# B&R Automation Studio project RTFProj (part 3)

#### Types.typ - Exported data types
```iecst
TYPE
	enum_opticalSensorInternal :
		(
		OS_INITIALIZATION := 0,
		OS_ENABLED := 1,
		OS_CALCULATION := 2,
		OS_ERROR := 3
		);
	struct_opticalSensorInternal : 	STRUCT
		index : ARRAY[0..1]OF USINT;
		auxiliary_pos : ARRAY[0..3]OF REAL;
		state : enum_opticalSensorInternal;
	END_STRUCT;
END_TYPE
```

#### ro_sensors.fun - Exported functions and function blocks
```iecst
FUNCTION err_modDetect : BOOL
	VAR_INPUT
		detect_err : ARRAY[0..3] OF BOOL;
		modul_ok : ARRAY[0..3] OF BOOL;
	END_VAR
	VAR
		i2 : USINT;
		i1 : USINT;
	END_VAR
END_FUNCTION

FUNCTION_BLOCK FB_DetectionPosition
	VAR_INPUT
		Enable : BOOL;
		Distance_Error : ARRAY[0..3] OF BOOL;
		Positions_FromTheSensors : ARRAY[0..3] OF REAL;
		Detection_Error : ARRAY[0..3] OF BOOL;
	END_VAR
	VAR_OUTPUT
		Actual_Positions : ARRAY[0..3] OF REAL;
		ModulOk : ARRAY[0..3] OF BOOL;
		Error : BOOL;
	END_VAR
	VAR
		Internal : struct_opticalSensorInternal;
	END_VAR
END_FUNCTION_BLOCK
```

#### FB_DetectionPosition.st
```iecst
FUNCTION_BLOCK FB_DetectionPosition

    IF Enable <> TRUE THEN
        // reset output variables
        Internal.index[0] := 0;
        Internal.index[1] := 0;

        Actual_Positions[0] := 0;
        Actual_Positions[1] := 0;
        Actual_Positions[2] := 0;
        Actual_Positions[3] := 0;

        ModulOk[0] := FALSE;
        ModulOk[1] := FALSE;
        ModulOk[2] := FALSE;
        ModulOk[3] := FALSE;

        Error := FALSE;

        // go to initialization state
        Internal.state := OS_INITIALIZATION;
    END_IF

    CASE Internal.state OF
        OS_INITIALIZATION:
            // INITIALIZATION STATE
            IF Enable = TRUE THEN
                Internal.state := OS_ENABLED;
            ELSE
                Internal.state := OS_INITIALIZATION;
            END_IF

        OS_ENABLED:
            // ENABLED STATE
            Error := err_modDetect(Detection_Error,ModulOk);

            IF Error = TRUE THEN
                Internal.state := OS_ERROR;
            ELSE
                Internal.state := OS_CALCULATION;
            END_IF

        OS_CALCULATION:
            // CALCULATION STATE
            FOR Internal.index[0] := 0 TO 3 DO
                IF Distance_Error[Internal.index[0]] = FALSE AND Internal.auxiliary_pos[Internal.index[0]] <> -9999 THEN
                    Internal.auxiliary_pos[Internal.index[0]] := 0;
                    Actual_Positions[Internal.index[0]]       := Positions_FromTheSensors[Internal.index[0]];
                ELSIF Distance_Error[Internal.index[0]] = TRUE AND Internal.auxiliary_pos[Internal.index[0]] <> -9999 THEN
                    Internal.auxiliary_pos[Internal.index[0]] := 0;
                    Actual_Positions[Internal.index[0]]       := -1000;
                ELSE
                    Actual_Positions[Internal.index[0]]       := Internal.auxiliary_pos[Internal.index[0]];
                    Internal.auxiliary_pos[Internal.index[0]] := 0;
                END_IF

            END_FOR

            Error := err_modDetect(Detection_Error,ModulOk);

            IF Error = TRUE THEN
                Internal.state := OS_ERROR;
            ELSE
                Internal.state := OS_CALCULATION;
            END_IF
        OS_ERROR:
            // ERROR STATE
            Error := err_modDetect(Detection_Error,ModulOk);

            IF Error = TRUE THEN
                FOR Internal.index[1] := 0 TO 3 DO
                    IF ModulOk[Internal.index[1]] = FALSE THEN
                        Internal.auxiliary_pos[Internal.index[1]] := -9999;
                    ELSE
                        Internal.auxiliary_pos[Internal.index[1]] := 0;
                    END_IF
                END_FOR

                Internal.state := OS_CALCULATION;
            ELSE
                Internal.state := OS_CALCULATION;
            END_IF
    END_CASE

END_FUNCTION_BLOCK

FUNCTION err_modDetect

    FOR i1 := 0 TO 3 DO
        IF detect_err[i1] = FALSE THEN
            modul_ok[i1] := TRUE;
        ELSE
            modul_ok[i1] := FALSE;
        END_IF
    END_FOR

    FOR i2 := 0 TO 3 DO
        IF modul_ok[i2] = FALSE THEN
            err_modDetect := TRUE;
            RETURN;
        ELSE
            err_modDetect := FALSE;
        END_IF
    END_FOR

END_FUNCTION
```

### Library Logical/Libraries/Camera (ANSIC)

#### Types.typ - Exported data types
```iecst
TYPE
	MainSwitch_enum :
		(
		DISABLED := 0,
		ENABLED := 1,
		RUN := 2,
		ERROR := 255
		);
	FTPSwitch_enum :
		(
		DEVLINK := 1,
		FILECOPY := 2,
		DEVUNLINK := 3
		);
	ControlSwitch_enum :
		(
		WAIT_CMD := 0,
		TRIGGER_RDY := 1,
		TRIGGER := 2,
		ACQ := 3,
		INSP := 4
		);
	InSight_type : 	STRUCT
		ModuleOk : BOOL;
		Control_I2000_S01 : UDINT; (*Camera control including trigger*)
		Status_I2001_S01 : UDINT;
		InspectionResults_I2011_S01 : UDINT; (*X Axis*)
		InspectionResults_I2011_S02 : UDINT; (*Y Axis*)
		InspectionResults_I2011_S03 : UDINT; (*Succes*)
		InspectionResults_I2011_S04 : UDINT; (*Fail*)
		UserData_I2021_S01 : UDINT; (*Change zone*)
	END_STRUCT;
	Internal_type : 	STRUCT
		NaN : REAL;
		CameraControl : CameraControl_type;
		MainSwitch : MainSwitch_enum;
		FTP : FTP_type;
		SuccesCount : UDINT;
		FailCount : UDINT;
		disableBit : USINT;
		Search_tmp : BOOL;
		Zone : Zone_enum;
		ChangeZone : ChangeZone_enum;
		oldState : ChangeZone_enum;
	END_STRUCT;
	Zone_enum :
		(
		ZONE1 := 0,
		ZONE2 := 1,
		ZONE3 := 2,
		ZONE4 := 3,
		ZONE5 := 4,
		ZONE6 := 5,
		ZONE7 := 6,
		ZONE8 := 7,
		WHOLE := 500
		);
	ChangeZone_enum :
		(
		CHANGE := 2,
		ONE_ZONE := 1,
		WHOLE_ZONE := 0
		);
	Results_type : 	STRUCT
		AxisX : REAL;
		AxisY : REAL;
		ActTime : RTCtime_typ;
		AxisXOld : REAL;
		AxisYOld : REAL;
		TimeDiff_ms : REAL;
		ActTimeOld : RTCtime_typ;
		NewVal : BOOL;
	END_STRUCT;
	CameraControl_type : 	STRUCT
		ControlSwitch : ControlSwitch_enum;
	END_STRUCT;
	MappView_type : 	STRUCT
		ZoneString : STRING[80];
		PicEnable : BOOL;
		Y : ARRAY[0..1000]OF INT;
		X : ARRAY[0..1000]OF INT := [11(5),0,996(0)];
		LoadImage : BOOL;
	END_STRUCT;
	FTP_type : 	STRUCT
		FileCopy_0 : FileCopy;
		DevLink_0 : DevLink;
		DevUnlink_0 : DevUnlink;
		Status : USINT;
		FTPSwitch : FTPSwitch_enum;
		pParam : STRING[200];
		handle : UDINT;
		pDevice : STRING[20];
		pDest : STRING[80];
		pSrc : STRING[80];
		pDestDev : STRING[20];
	END_STRUCT;
END_TYPE
```

#### Constants.var - Exported constants
```iecst
VAR CONSTANT
	ERR_OK : UINT := 0;
	FB_DISABLED : UINT := 65534; (*Function block is disabled*)
	ERR_CAM_NOTFOUND : UINT := 65533; (*Camera not found*)
	ERR_FTP_NOTREADY : UINT := 62687; (*FTP not ready*)
END_VAR
```

#### Camera.fun - Exported functions and function blocks
```iecst
FUNCTION_BLOCK FBCamera
	VAR_INPUT
		Enable : BOOL;
		InSight : InSight_type;
		ErrorReset : BOOL;
		Search : BOOL;
	END_VAR
	VAR_OUTPUT
		Active : BOOL;
		Error : BOOL;
		Status : UINT;
		isCameraReady : BOOL;
		isSearching : BOOL;
		isBallFound : BOOL;
		Results : Results_type;
	END_VAR
	VAR
		Internal : Internal_type;
	END_VAR
END_FUNCTION_BLOCK
```

#### Camera.c
```c
#include <bur/plctypes.h>
#include <math.h>

#ifdef _DEFAULT_INCLUDES
#include <AsDefault.h>
#endif

#define NaN sqrt(-1)
#define CAM_OFFLINE_MASK 128												//1000 0000b
#define CAM_ONLINE_MASK 0xFFFFFF7F

#define CAM_USER_DATA 0x10004												//Mask for user data ack
#define CAM_FIND_WHOLE_ZONE 0xFFFFFFFF										//Mask for finding at whole playground

#define MAX_DIFF_PER 0.15													//Max diffrence between old and actual value in %

#define ABS_F(X) ((X) < (0) ? -(X) : (X)) 									//ABS funkcion
							//		  |							9800
#define X1_REF_PLGND 800.0	//(UNITS) |				   3800 6800  | 11300
#define X2_REF_PLGND 11300.0//(UNITS) |				 _____|___|___|_|_
#define X1_REF_CAM 1215.0	//(PIXELS)|				| | | O O O O | | |		SCHEME OF X AXIS
#define X2_REF_CAM 82.0		//(PIXELS)|				| | O | O O | O | |		AND PLAYGROUND WITH
 							//		  |		    	| O | O O O O | O |		DISTANCE OF PLAYERS
#define Y1_REF_PLGND 820.0	//(UNITS) |	 	  		| | O | O O | O | |		IN UNITS
#define Y2_REF_PLGND -950.0 //(UNITS) |				|_|_|_O_O_O_O_|_|_|		(10 UNITS = 1 MM)
#define Y1_REF_CAM 414.0	//(PIXELS)| 		      | |   |   |
#define Y2_REF_CAM 604.0	//(PIXELS)|			 	800 | 5300 8300
							//		  |		    	   2300

#define X_LIN_EQ_K ((X1_REF_PLGND-X2_REF_PLGND)/(X1_REF_CAM-X2_REF_CAM)) 		//Define K-parameter of line equaton for X axis
#define X_LIN_EQ_Q (X1_REF_PLGND-(X1_REF_CAM*X_LIN_EQ_K))				 		//Define Q-parameter of line equaion for X axis

#define Y_LIN_EQ_K ((Y1_REF_PLGND-Y2_REF_PLGND)/(Y1_REF_CAM-Y2_REF_CAM))		//Define K-parameter of line equaton for Y axis
#define Y_LIN_EQ_Q (Y1_REF_PLGND-(Y1_REF_CAM*Y_LIN_EQ_K))						//Define Q-parameter of line equaton for Y axis

#define X_MAX_DIFF ABS_F((X_LIN_EQ_K+X_LIN_EQ_Q)-((2*X_LIN_EQ_K)+X_LIN_EQ_Q))	//Line equation for X axis
#define Y_MAX_DIFF ABS_F((Y_LIN_EQ_K+Y_LIN_EQ_Q)-((2*Y_LIN_EQ_K)+Y_LIN_EQ_Q))	//Line equation for Y axis

void setError(struct FBCamera *inst,unsigned int status);
void initFB(struct FBCamera *inst);
void resetFB(struct FBCamera *inst);
void getRealAxes(struct FBCamera *inst);
void cleanFB(struct FBCamera *inst);
REAL RctToReal_ms (struct RTCtime_typ RTCtime);

void FBCamera(struct FBCamera *inst)
{
	if ((!inst->Enable) && (!inst->Internal.disableBit))
		cleanFB(inst);

	switch (inst->Internal.MainSwitch){										//Main switch, DISABLED FB, INITialising FB, ENABLED FB and ERROR case
		/******************************************************************/
		/*							FB is DISABLED					 	  */
		/******************************************************************/

		case DISABLED:														//FB is disabled
			if (inst->Internal.disableBit){
				cleanFB(inst);
				inst->Internal.disableBit = 1;
			}
			if (inst->Enable){												//Wait for Enable = TRUE, else do nothing
				inst->Internal.MainSwitch = ENABLED;						//Go to ENABLED case
				inst->Internal.disableBit = 0;
			}
			else
				inst->Status = ERR_FUB_ENABLE_FALSE;						//Status 65534, FB is called but not enabled
			break;

		/******************************************************************/
		/*				FB is ENABLED but Camera is not ready		 	  */
		/******************************************************************/

		case ENABLED:														//FB is enabled and working
			inst->Status = ERR_OK;											//No error in enable case
			inst->Active = 1;												//variable indicating active FB
			if (!inst->InSight.ModuleOk){									//InSight Camera is not connected properly
				inst->isCameraReady = 0;									//Bit for user that Camera is not working
				if (inst->Search)											//If user allow searching for ball, change case to ERROR because you cannot find while there is no camera
					setError(inst,ERR_CAM_NOTFOUND);						//Error, Status 65533 - camera not found
			}
			else {
				inst->isCameraReady = 1;									//Bit for user that Camera is working
				inst->Internal.MainSwitch = RUN;							//Change state to RUN
			}
			break;

		/******************************************************************/
		/*						FB and Camera are ready				 	  */
		/******************************************************************/
		case RUN:															//FB is enabled and camera communicating
			if (!(inst->InSight.ModuleOk))									//if camera is disconnected change state to ENABLE where waiting for connect
				inst->Internal.MainSwitch = ENABLED;
			if (inst->Search){
				inst->isSearching = 1;
				inst->InSight.Control_I2000_S01 &= CAM_ONLINE_MASK;			//Disable control bit for cammera offline mode
				switch (inst->Internal.ChangeZone){
					case CHANGE:
						if ((inst->InSight.Control_I2000_S01 & CAM_USER_DATA) == CAM_USER_DATA){
							if ((inst->InSight.Status_I2001_S01 & 0x10000) == 0x10000) {
								if (inst->Internal.oldState == ONE_ZONE)
									inst->Internal.ChangeZone = WHOLE_ZONE;
								else
									inst->Internal.ChangeZone = ONE_ZONE;
								inst->InSight.Control_I2000_S01 &= 0xFFFEFFFB;
							}
						}
						else inst->Internal.ChangeZone = WHOLE_ZONE;
						break;

					case ONE_ZONE:
						getRealAxes(inst);
						inst->Internal.oldState = ONE_ZONE;
						if (((isnan(inst->Results.AxisX)) || isnan(inst->Results.AxisY)) && (inst->Results.NewVal)){
							inst->Internal.ChangeZone = CHANGE;
							inst->InSight.Control_I2000_S01 |= CAM_USER_DATA;
							inst->InSight.UserData_I2021_S01 = 65535;
						}
						switch (inst->Internal.Zone){
							case ZONE1:
								strcpy(inst->MappView.ZoneString,"Zone 1");
								break;

							case ZONE2:
								strcpy(inst->MappView.ZoneString,"Zone 2");
								break;

							case ZONE3:
								strcpy(inst->MappView.ZoneString,"Zone 3");
								break;

							case ZONE4:
								strcpy(inst->MappView.ZoneString,"Zone 4");
								break;

							case ZONE5:
								strcpy(inst->MappView.ZoneString,"Zone 5");
								break;

							case ZONE6:
								strcpy(inst->MappView.ZoneString,"Zone 6");
								break;

							case ZONE7:
								strcpy(inst->MappView.ZoneString,"Zone 7");
								break;

							case WHOLE:

								break;
						}
						break;

					case WHOLE_ZONE:
						getRealAxes(inst);
						inst->Internal.Zone = WHOLE;
						inst->Internal.oldState = WHOLE_ZONE;
						strcpy(inst->MappView.ZoneString,"Whole");
						if(inst->isBallFound){
							inst->Internal.ChangeZone = CHANGE;
							inst->InSight.Control_I2000_S01 |= CAM_USER_DATA;
							if (inst->Results.AxisX > 10300){
								inst->InSight.UserData_I2021_S01 = 1;
								inst->Internal.Zone = ZONE1;}
							else if (inst->Results.AxisX > 9050){
								inst->InSight.UserData_I2021_S01 = 2;
								inst->Internal.Zone = ZONE2;}
							else if (inst->Results.AxisX > 7350){
								inst->InSight.UserData_I2021_S01 = 4;
								inst->Internal.Zone = ZONE3;}
							else if (inst->Results.AxisX > 6250){
								inst->InSight.UserData_I2021_S01 = 8;
								inst->Internal.Zone = ZONE4;}
							else if (inst->Results.AxisX > 4400){
								inst->InSight.UserData_I2021_S01 = 16;
								inst->Internal.Zone = ZONE5;}
							else if (inst->Results.AxisX > 2460){
								inst->InSight.UserData_I2021_S01 = 32;
								inst->Internal.Zone = ZONE6;}
							else if (inst->Results.AxisX > 0){
								inst->InSight.UserData_I2021_S01 = 64;
								inst->Internal.Zone = ZONE7;}
							else{
								inst->Internal.ChangeZone = WHOLE_ZONE;
								inst->InSight.Control_I2000_S01 &= 0xFFFEFFFB;
								inst->InSight.UserData_I2021_S01 = 0xFFFF;
							}
						}
						break;

				}
			}
			else{
				inst->InSight.Control_I2000_S01 |= CAM_OFFLINE_MASK;
				inst->isSearching = 0;
			}
			break;

		case ERROR:															//error case, to change state is needed error Reset variable or disable FB
			inst->Error = 1;												//Change Error variable
			inst->Internal.CameraControl.ControlSwitch = WAIT_CMD;			//Reset camera trigger state
			inst->isSearching = 0;											//FB cannot searching in error case
			if (inst->ErrorReset){											//waiting on ErrorReset
				inst->Error = 0;
				inst->Status = ERR_OK;
				resetFB(inst);
				inst->Internal.MainSwitch = ENABLED;						//change state
			}
			break;
	}

	if (inst->ErrorReset)
		resetFB(inst);

	if (inst->Error == 1)
		inst->Internal.MainSwitch = ERROR;

}

void initFB(struct FBCamera *inst)
{
	inst->Active = 0;
	inst->Error = 0;
	inst->ErrorReset = 0;
	inst->isCameraReady = 0;
	inst->isBallFound = 0;
	inst->isSearching = 0;
	inst->Search = 0;
	inst->Status = ERR_OK;
	inst->Internal.CameraControl.ControlSwitch = WAIT_CMD;
	inst->Internal.MainSwitch = DISABLED;
	inst->Internal.Search_tmp = 0;
	inst->Internal.disableBit = 1;
	inst->InSight.Control_I2000_S01 |= CAM_OFFLINE_MASK;
	memset(&inst->Results.ActTime,0,sizeof(inst->Results.ActTime));
	inst->Results.AxisXOld = NaN;
	inst->Results.AxisYOld = NaN;
	inst->InSight.Control_I2000_S01 |= CAM_USER_DATA;
	inst->InSight.UserData_I2021_S01 = 65535;
	inst->Internal.ChangeZone = CHANGE;
}

void resetFB(struct FBCamera *inst)
{
	inst->ErrorReset = 0;							//Reset error reset
	inst->Error = 0;								//Reset Error
	inst->Status = ERR_OK;
}

void cleanFB(struct FBCamera *inst)
{
	initFB(inst);
	resetFB(inst);
}

void setError(struct FBCamera *inst,unsigned int status) {
	inst->Error = 1;
	inst->Status = status;
}

void getRealAxes(struct FBCamera *inst)
{
	if (inst->Internal.SuccesCount != inst->InSight.InspectionResults_I2011_S03){
		inst->Results.NewVal = 1;
		REAL AxisXnew = ((inst->InSight.InspectionResults_I2011_S01*X_LIN_EQ_K)+X_LIN_EQ_Q);
		REAL AxisYnew = ((inst->InSight.InspectionResults_I2011_S02*Y_LIN_EQ_K)+Y_LIN_EQ_Q);

		if (((AxisXnew >= 0) && (AxisXnew < 12100)) && ((AxisYnew < 3515) && (AxisYnew > -3515))){

			if (isnan(inst->Results.AxisX) || isnan(inst->Results.AxisY)){
				inst->Results.AxisX = AxisXnew;
				inst->Results.AxisY = AxisYnew;
			}
			else if(((ABS_F(AxisXnew - (inst->Results.AxisX))) < (X_MAX_DIFF * 2)) && (((ABS_F(AxisYnew - (inst->Results.AxisY))) < (Y_MAX_DIFF * 2)))) {
				inst->Results.AxisXOld = inst->Results.AxisX = ((AxisXnew + inst->Results.AxisX)/2);
				inst->Results.AxisYOld = inst->Results.AxisY = ((AxisYnew + inst->Results.AxisY)/2);
			}
			else{
				inst->Results.AxisXOld = inst->Results.AxisX;
				inst->Results.AxisYOld = inst->Results.AxisY;
				inst->Results.AxisX = AxisXnew;
				inst->Results.AxisY = AxisYnew;
			}
			memcpy((UDINT)&inst->Results.ActTimeOld,(UDINT)&inst->Results.ActTime,sizeof(inst->Results.ActTime));
			RTC_gettime(&inst->Results.ActTime);
			inst->Results.TimeDiff_ms = ((RctToReal_ms(inst->Results.ActTime)) - (RctToReal_ms(inst->Results.ActTimeOld)));
			inst->isBallFound = 1;
			inst->Status = ERR_OK;
			inst->Internal.SuccesCount = inst->InSight.InspectionResults_I2011_S03;
		}
		else{
			inst->Status = ERR_BALL_OUTRANGE;
			inst->isBallFound = 0;
		}
	}
	else if (inst->Internal.FailCount != inst->InSight.InspectionResults_I2011_S04){
		inst->Results.NewVal = 1;
		if (!isnan(inst->Results.AxisX) || !isnan(inst->Results.AxisY)){
			inst->Results.AxisXOld = inst->Results.AxisX;
			inst->Results.AxisYOld = inst->Results.AxisY;
		}
		inst->Results.AxisX = inst->Results.AxisY = NaN;
		inst->Internal.FailCount = inst->InSight.InspectionResults_I2011_S04;
		inst->isBallFound = 0;
		memcpy((UDINT)&inst->Results.ActTimeOld,(UDINT)&inst->Results.ActTime,sizeof(inst->Results.ActTime));
		RTC_gettime(&inst->Results.ActTime);
		inst->Results.TimeDiff_ms = ((RctToReal_ms(inst->Results.ActTime)) - (RctToReal_ms(inst->Results.ActTimeOld)));
	}
	else{
		inst->isBallFound = 0;
		inst->Results.NewVal = 1;
	}
}

REAL RctToReal_ms (struct RTCtime_typ RTCtime){
	return(((REAL)RTCtime.hour*3600000)+((REAL)RTCtime.minute*60000)+((REAL)RTCtime.second*1000)+((REAL)RTCtime.millisec)+((REAL)RTCtime.microsec/1000));
}
```

### Library Logical/Libraries/Bar_Light (ANSIC)

#### Bar_light.c
```c
#include <bur/plctypes.h>
#include <MTBasics.h>
#include <brsystem.h>
#include <math.h>

#ifdef _DEFAULT_INCLUDES
#include <AsDefault.h>
#endif

void resetFB(struct Light *inst);												//Reset basic variables
void PWMControl(struct Light *inst);											//Controls Light in PWM Mode
void BlinkControl(struct Light *inst);											//Allows Blinking of Light

void Light(struct Light *inst)
{
	if ((!inst->Enable) && (inst->internal.MainControlBarLight != INIT_BARLIGHT))//If FB not allowed and switch is not in init state
		inst->internal.MainControlBarLight = DISABLED_BARLIGHT;					//Change state to DISABLED

	switch (inst->internal.MainControlBarLight)									//Main switch controls whole FB
	{
		case INIT_BARLIGHT:														//Check parameter for PWM
			inst->internal.TaskClass.RTInfo_0.enable = 1;
			RTInfo(&inst->internal.TaskClass.RTInfo_0);
			if (!(inst->internal.TaskClass.RTInfo_0.status) && (inst->internal.TaskClass.RTInfo_0.cycle_time > 0))
			{
				if (inst->internal.TaskClass.RTInfo_0.cycle_time <= 1000)
				{
					inst->isPWMEnabled = inst->internal.PWM.PWMEnabled = 1;
					inst->isPWMEnabled = inst->internal.PWM.PWM.Enable = 1;
					inst->internal.PWM.PWM.MinPulseWidth = 0.001;
					inst->internal.PWM.PWM.Period = 0.01;
					inst->internal.PWM.PWM.Mode = mtBASICS_PULSE_BEGINNING;
				}
				else
					inst->isPWMEnabled = inst->internal.PWM.PWMEnabled = 0;

				inst->internal.PWM.PWM.DutyCycle = 100;
				inst->internal.TaskClass.RTInfo_0.enable = 0;
				inst->internal.TaskClass.CyclicTime = ((inst->internal.TaskClass.RTInfo_0.cycle_time)/1000);
				inst->internal.MainControlBarLight = DISABLED_BARLIGHT;
			}
			break;

		case DISABLED_BARLIGHT:
			if (inst->Enable)
			{
				if (inst->DO9322.ModuleOK)
				{
					inst->internal.MainControlBarLight = ENABLED_BARLIGHT;
					resetFB(inst);
				}
				else
				{
					inst->Status = DO9322_NOT_CONNECTED;
					inst->internal.MainControlBarLight = ERROR_BARLIGHT;
				}
			}
			break;

		case ENABLED_BARLIGHT:
			inst->Active = 1;
			if (inst->PowerOn)
			{
				if (inst->Blinking.StartBlinking)
				{
					BlinkControl(inst);
				}
				else if (inst->internal.PWM.PWMEnabled)
				{
					PWMControl(inst);
				}
				else inst->DO9322.DigitalOutput = 1;
			}
			else inst->DO9322.DigitalOutput = 0;
			break;

		case ERROR_BARLIGHT:
			inst->Error = 1;
			break;
	}
}

void resetFB(struct Light *inst)
{
	inst->Active = 0;
	inst->Blinking.StartBlinking = 0;
	inst->DO9322.DigitalOutput = 0;
	inst->DutyCycle = 100;
	inst->Error = 0;
	inst->PowerOn = 0;
	inst->isPowerOn = 0;
	inst->Status = ERR_OK;
}

void PWMControl(struct Light *inst)
{
	inst->internal.PWM.PWM.DutyCycle = inst->DutyCycle;
	MTBasicsPWM(&inst->internal.PWM.PWM);
	inst->DO9322.DigitalOutput = inst->internal.PWM.PWM.Out;
}

void BlinkControl(struct Light *inst)
{
	inst->internal.BlinkingCounter += 1;
	if ((inst->internal.BlinkingCounter*inst->internal.TaskClass.CyclicTime) < inst->Blinking.BlinkingTime_ms)
	{
		if ((inst->internal.BlinkCounter*inst->internal.TaskClass.CyclicTime) >= inst->Blinking.BlinkPeriod_ms)
		{
			inst->DO9322.DigitalOutput = !inst->DO9322.DigitalOutput;
			inst->internal.BlinkCounter = 0;
		}
		else
		{
			inst->internal.BlinkCounter += 1;
		}
	}
	else
	{
		inst->internal.BlinkingCounter = 0;
		inst->internal.BlinkCounter = 0;
		inst->DO9322.DigitalOutput = 0;
		inst->Blinking.StartBlinking = 0;
	}
}
```

### Library Logical/Libraries/LB_Camera/Camera (ANSIC)

#### Camera.c
```c
#include <bur/plctypes.h>
#include <math.h>

#ifdef _DEFAULT_INCLUDES
#include <AsDefault.h>
#endif

#define NaN sqrt(-1)
#define CAM_OFFLINE_MASK 128												//1000 0000b
#define CAM_ONLINE_MASK 0xFFFFFF7F

#define ABS_F(X) ((X) < (0) ? -(X) : (X)) 									//ABS funkcion
							//		  |							9800
#define X1_REF_PLGND 800.0	//(UNITS) |				   3800 6800  | 11300
#define X2_REF_PLGND 11300.0//(UNITS) |				 _____|___|___|_|_
#define X1_REF_CAM 1215.0	//(PIXELS)|				| | | O O O O | | |		SCHEME OF X AXIS
#define X2_REF_CAM 82.0		//(PIXELS)|				| | O | O O | O | |		AND PLAYGROUND WITH
 							//		  |		    	| O | O O O O | O |		DISTANCE OF PLAYERS
#define Y1_REF_PLGND 820.0	//(UNITS) |	 	  		| | O | O O | O | |		IN UNITS
#define Y2_REF_PLGND -950.0 //(UNITS) |				|_|_|_O_O_O_O_|_|_|		(10 UNITS = 1 MM)
#define Y1_REF_CAM 414.0	//(PIXELS)| 		      | |   |   |
#define Y2_REF_CAM 604.0	//(PIXELS)|			 	800 | 5300 8300
							//		  |		    	   2300

#define X_LIN_EQ_K ((X1_REF_PLGND-X2_REF_PLGND)/(X1_REF_CAM-X2_REF_CAM)) 		//Define K-parameter of line equaton for X axis
#define X_LIN_EQ_Q (X1_REF_PLGND-(X1_REF_CAM*X_LIN_EQ_K))				 		//Define Q-parameter of line equaion for X axis

#define Y_LIN_EQ_K ((Y1_REF_PLGND-Y2_REF_PLGND)/(Y1_REF_CAM-Y2_REF_CAM))		//Define K-parameter of line equaton for Y axis
#define Y_LIN_EQ_Q (Y1_REF_PLGND-(Y1_REF_CAM*Y_LIN_EQ_K))						//Define Q-parameter of line equaton for Y axis

#define X_MAX_DIFF ABS_F((X_LIN_EQ_K+X_LIN_EQ_Q)-((2*X_LIN_EQ_K)+X_LIN_EQ_Q))	//Line equation for X axis
#define Y_MAX_DIFF ABS_F((Y_LIN_EQ_K+Y_LIN_EQ_Q)-((2*Y_LIN_EQ_K)+Y_LIN_EQ_Q))	//Line equation for Y axis

void setError(struct FBCamera *inst,unsigned int status);
void initFB(struct FBCamera *inst);
void resetFB(struct FBCamera *inst);
void getRealAxes(struct FBCamera *inst);
void cleanFB(struct FBCamera *inst);
REAL RctToReal_ms (struct RTCtime_typ RTCtime);

void FBCamera(struct FBCamera *inst)
{
	if ((!inst->Enable) && (!inst->Internal.disableBit))
		cleanFB(inst);

	switch (inst->Internal.MainSwitch){										//Main switch, DISABLED FB, INITialising FB, ENABLED FB and ERROR case
		/******************************************************************/
		/*							FB is DISABLED					 	  */
		/******************************************************************/

		case DISABLED:														//FB is disabled
			if (inst->Internal.disableBit){
				cleanFB(inst);
				inst->Internal.disableBit = 1;
			}
			if (inst->Enable){												//Wait for Enable = TRUE, else do nothing
				inst->Internal.MainSwitch = ENABLED;						//Go to ENABLED case
				inst->Internal.disableBit = 0;
			}
			else
				inst->Status = ERR_FUB_ENABLE_FALSE;						//Status 65534, FB is called but not enabled
			break;

		/******************************************************************/
		/*				FB is ENABLED but Camera is not ready		 	  */
		/******************************************************************/

		case ENABLED:														//FB is enabled and working
			inst->Active = 1;												//variable indicating active FB
			if (!inst->InSight.ModuleOk){									//InSight Camera is not connected properly
				inst->isCameraReady = 0;									//Bit for user that Camera is not working
				if (inst->Search)											//If user allow searching for ball, change case to ERROR because you cannot find while there is no camera
					setError(inst,ERR_CAM_NOTFOUND);						//Error, Status 65533 - camera not found
			}
			else {
				unsigned int status;
				inst->isCameraReady = 1;								//Bit for user that Camera is working
				inst->Internal.MainSwitch = RUN;						//Change state to RUN
				inst->Status = ERR_OK;									//No error in enable case
			}
			break;

		case RUN:															//FB is enabled and camera communicating
			if (!(inst->InSight.ModuleOk))									//if camera is disconnected change state to ENABLE where waiting for connect
				inst->Internal.MainSwitch = ENABLED;
			if (inst->Search){
				inst->InSight.Control_I2000_S01 &= CAM_ONLINE_MASK;			//Disable control bit for cammera offline mode
				inst->isSearching = 1;
				if (inst->InSight.InspectionResults_I2011_S03 != inst->Internal.SuccesCount)
					inst->isBallFound = 1;
				else inst->isBallFound = 0;
				getRealAxes(inst);
			}
			else{
				inst->InSight.Control_I2000_S01 |= CAM_OFFLINE_MASK;
				inst->isSearching = 0;
			}
			break;

		case ERROR:															//error case, to change state is needed error Reset variable or disable FB
			inst->Error = 1;												//Change Error variable
			inst->Internal.CameraControl.ControlSwitch = WAIT_CMD;			//Reset camera trigger state
			inst->isSearching = 0;											//FB cannot searching in error case
			if (inst->ErrorReset){											//waiting on ErrorReset
				inst->Error = 0;
				inst->Status = ERR_OK;
				resetFB(inst);
				inst->Internal.MainSwitch = ENABLED;						//change state
			}
			break;
	}

	if (inst->ErrorReset)
		resetFB(inst);

	if (inst->Error == 1)
		inst->Internal.MainSwitch = ERROR;

}

void initFB(struct FBCamera *inst)
{
	inst->Active = 0;
	inst->Error = 0;
	inst->ErrorReset = 0;
	inst->isCameraReady = 0;
	inst->isBallFound = 0;
	inst->isSearching = 0;
	inst->Search = 0;
	inst->Status = ERR_OK;
	inst->Internal.CameraControl.ControlSwitch = WAIT_CMD;
	inst->Internal.MainSwitch = DISABLED;
	inst->Internal.Search_tmp = 0;
	inst->Internal.disableBit = 1;
	inst->InSight.Control_I2000_S01 |= CAM_OFFLINE_MASK;
	memset(&inst->Results.ActTime,0,sizeof(inst->Results.ActTime));
	inst->Results.AxisXOld = NaN;
	inst->Results.AxisYOld = NaN;
}

void resetFB(struct FBCamera *inst)
{
	inst->ErrorReset = 0;							//Reset error reset
	inst->Error = 0;								//Reset Error
	inst->Status = ERR_OK;
}

void cleanFB(struct FBCamera *inst)
{
	initFB(inst);
	resetFB(inst);
}

void setError(struct FBCamera *inst,unsigned int status) {
	inst->Error = 1;
	inst->Status = status;
}

void getRealAxes(struct FBCamera *inst)
{
	if (inst->Internal.SuccesCount != inst->InSight.InspectionResults_I2011_S03){
		if(((ABS_F(((inst->InSight.InspectionResults_I2011_S01*X_LIN_EQ_K)+X_LIN_EQ_Q)-(inst->Results.AxisX))) < (X_MAX_DIFF + (0.1*X_MAX_DIFF))) &&
		((ABS_F(((inst->InSight.InspectionResults_I2011_S02*Y_LIN_EQ_K)+Y_LIN_EQ_Q)-(inst->Results.AxisY))) < (Y_MAX_DIFF + (0.1*Y_MAX_DIFF)))) {
			inst->Results.AxisX = ((((inst->InSight.InspectionResults_I2011_S01*(X_LIN_EQ_K))+X_LIN_EQ_Q)+inst->Results.AxisX)/2);
			inst->Results.AxisY = ((((inst->InSight.InspectionResults_I2011_S02*(Y_LIN_EQ_K))+Y_LIN_EQ_Q)+inst->Results.AxisY)/2);
			inst->Results.AxisXOld = inst->Results.AxisYOld = NaN;
		}
		else{
			inst->Results.AxisXOld = inst->Results.AxisX;
			inst->Results.AxisYOld = inst->Results.AxisY;
			inst->Results.AxisX = ((inst->InSight.InspectionResults_I2011_S01*(X_LIN_EQ_K))+X_LIN_EQ_Q);
			inst->Results.AxisY = ((inst->InSight.InspectionResults_I2011_S02*(Y_LIN_EQ_K))+Y_LIN_EQ_Q);

		}
		memcpy((UDINT)&inst->Results.ActTimeOld,(UDINT)&inst->Results.ActTime,sizeof(inst->Results.ActTime));
		RTC_gettime(&inst->Results.ActTime);
		inst->Results.TimeDiff_ms = ((RctToReal_ms(inst->Results.ActTime)) - (RctToReal_ms(inst->Results.ActTimeOld)));
		inst->isBallFound = 1;
		inst->Internal.SuccesCount = inst->InSight.InspectionResults_I2011_S03;
	}
	else if ((inst->Internal.FailCount != inst->InSight.InspectionResults_I2011_S04) && ((!isnan(inst->Results.AxisXOld)) && (!isnan(inst->Results.AxisYOld)))){
		inst->Results.AxisX = inst->Results.AxisXOld;
		inst->Results.AxisY = inst->Results.AxisYOld;
		inst->Results.AxisXOld = inst->Results.AxisYOld = NaN;
		inst->Internal.FailCount = inst->InSight.InspectionResults_I2011_S04;
		inst->isBallFound = 0;
	}
}

REAL RctToReal_ms (struct RTCtime_typ RTCtime){
	return(((REAL)RTCtime.hour*3600000)+((REAL)RTCtime.minute*60000)+((REAL)RTCtime.second*1000)+((REAL)RTCtime.millisec)+((REAL)RTCtime.microsec/1000));
}
```

#### Types.typ - Exported data types
```iecst
TYPE
	MainSwitch_enum :
		(
		DISABLED := 0,
		ENABLED := 1,
		RUN := 2,
		ERROR := 255
		);
	FTPSwitch_enum :
		(
		DEVLINK := 1,
		FILECOPY := 2,
		DEVUNLINK := 3
		);
	ControlSwitch_enum :
		(
		WAIT_CMD := 0,
		TRIGGER_RDY := 1,
		TRIGGER := 2,
		ACQ := 3,
		INSP := 4
		);
	InSight_type : 	STRUCT
		ModuleOk : BOOL;
		Control_I2000_S01 : UDINT; (*Camera control including trigger*)
		Status_I2001_S01 : UDINT;
		InspectionResults_I2011_S02 : UDINT;
		InspectionResults_I2011_S01 : UDINT;
	END_STRUCT;
	Internal_type : 	STRUCT
		NaN : REAL;
		CameraControl : CameraControl_type;
		MainSwitch : MainSwitch_enum;
		FTP : FTP_type;
		disableBit : USINT;
		Search_tmp : BOOL;
	END_STRUCT;
	Results_type : 	STRUCT
		AxisX : REAL;
		AxisY : REAL;
		ActTime : RTCtime_typ;
		AxisXOld : REAL;
		AxisYOld : REAL;
		TimeDiff : REAL;
		ActTimeOld : RTCtime_typ;
	END_STRUCT;
	CameraControl_type : 	STRUCT
		ControlSwitch : ControlSwitch_enum;
	END_STRUCT;
	MappView_type : 	STRUCT
		PicEnable : BOOL;
		Y : ARRAY[0..1000]OF INT;
		X : ARRAY[0..1000]OF INT := [11(5),0,996(0)];
		LoadImage : BOOL;
	END_STRUCT;
	FTP_type : 	STRUCT
		FileCopy_0 : FileCopy;
		DevLink_0 : DevLink;
		DevUnlink_0 : DevUnlink;
		Status : USINT;
		FTPSwitch : FTPSwitch_enum;
		pParam : STRING[200];
		handle : UDINT;
		pDevice : STRING[20];
		pDest : STRING[80];
		pSrc : STRING[80];
		pDestDev : STRING[20];
	END_STRUCT;
END_TYPE
```

#### Constants.var - Exported constants
```iecst
VAR CONSTANT
	ERR_OK : UINT := 0;
	FB_DISABLED : UINT := 65534; (*Function block is disabled*)
	ERR_CAM_NOTFOUND : UINT := 65533; (*Camera not found*)
END_VAR
```

### Library Logical/Libraries/LB_Camera/Bar_Light (ANSIC)
Depends on: MTBasics, brsystem

#### Bar_light.c
```c
#include <bur/plctypes.h>
#include <MTBasics.h>
#include <brsystem.h>
#include <math.h>

#ifdef _DEFAULT_INCLUDES
#include <AsDefault.h>
#endif

void resetFB(struct Light *inst);
void PWMControl(struct Light *inst);
void BlinkControl(struct Light *inst);

void Light(struct Light *inst)
{
	if ((!inst->Enable) && (inst->internal.MainControlBarLight != INIT_BARLIGHT))
	{
		inst->internal.MainControlBarLight = DISABLED_BARLIGHT;
	}

	switch (inst->internal.MainControlBarLight)
	{
		case INIT_BARLIGHT:
			inst->internal.TaskClass.RTInfo_0.enable = 1;
			RTInfo(&inst->internal.TaskClass.RTInfo_0);
			if (!(inst->internal.TaskClass.RTInfo_0.status) && (inst->internal.TaskClass.RTInfo_0.cycle_time > 0))
			{
				if (inst->internal.TaskClass.RTInfo_0.cycle_time <= 1000)
				{
					inst->isPWMEnabled = inst->internal.PWM.PWMEnabled = 1;
					inst->internal.PWM.PWM.MinPulseWidth = 0.001;
					inst->internal.PWM.PWM.Period = 0.1;
					inst->internal.PWM.PWM.Mode = mtBASICS_PULSE_BEGINNING;
				}
				else
					inst->isPWMEnabled = inst->internal.PWM.PWMEnabled = 0;

				inst->internal.PWM.PWM.DutyCycle = 100;
				inst->internal.TaskClass.RTInfo_0.enable = 0;
				inst->internal.TaskClass.CyclicTime = ((inst->internal.TaskClass.RTInfo_0.cycle_time)/1000);
				inst->internal.MainControlBarLight = DISABLED_BARLIGHT;
			}
			break;

		case DISABLED_BARLIGHT:
			if (inst->Enable)
			{
				if (inst->DO9322.ModuleOK)
				{
					inst->internal.MainControlBarLight = ENABLED_BARLIGHT;
					resetFB(inst);
				}
				else
				{
					inst->Status = DO9322_NOT_CONNECTED;
					inst->internal.MainControlBarLight = ERROR_BARLIGHT;
				}
			}
			break;

		case ENABLED_BARLIGHT:
			inst->Active = 1;
			if (inst->PowerOn)
			{
				if (inst->Blinking.StartBlinking)
				{
					BlinkControl(inst);
				}
				else if (inst->internal.PWM.PWMEnabled)
				{
					PWMControl(inst);
				}
				else inst->DO9322.DigitalOutput = 1;
			}
			else inst->DO9322.DigitalOutput = 0;
			break;

		case ERROR_BARLIGHT:
			inst->Error = 1;
			break;
	}
}

void resetFB(struct Light *inst)
{
	inst->Active = 0;
	inst->Blinking.StartBlinking = 0;
	inst->DO9322.DigitalOutput = 0;
	inst->DutyCycle = 100;
	inst->Error = 0;
	inst->PowerOn = 0;
	inst->isPowerOn = 0;
	inst->Status = ERR_OK;
}

void PWMControl(struct Light *inst)
{
	MTBasicsPWM(&inst->internal.PWM.PWM);
	inst->DO9322.DigitalOutput = inst->internal.PWM.PWM.Out;
}

void BlinkControl(struct Light *inst)
{
	inst->internal.BlinkingCounter += 1;
	if ((inst->internal.BlinkingCounter*inst->internal.TaskClass.CyclicTime) < inst->Blinking.BlinkingTime_ms)
	{
		if ((inst->internal.BlinkCounter*inst->internal.TaskClass.CyclicTime) >= inst->Blinking.BlinkPeriod_ms)
		{
			inst->DO9322.DigitalOutput = !inst->DO9322.DigitalOutput;
			inst->internal.BlinkCounter = 0;
		}
		else
		{
			inst->internal.BlinkCounter += 1;
		}
	}
	else
	{
		inst->internal.BlinkingCounter = 0;
		inst->internal.BlinkCounter = 0;
		inst->DO9322.DigitalOutput = 0;
		inst->Blinking.StartBlinking = 0;
	}
}
```

### Data object Logical/ACP10_ETXEN/acp10etxen (Ett)

- acp10etxen.ett (not shown)


- Data object Logical/Simulation/Motion/dfRotSobj/dfRotSa (Apt) (no source held here)

- Data object Logical/Simulation/Motion/dfRotSobj/dfRotSi (Ax) (no source held here)

- Data object Logical/Simulation/Motion/gkRotSobj/gkRotSa (Apt) (no source held here)

- Data object Logical/Simulation/Motion/gkRotSobj/gkRotSi (Ax) (no source held here)

- Data object Logical/Simulation/Motion/dfLinSobj/dfLinSa (Apt) (no source held here)

- Data object Logical/Simulation/Motion/dfLinSobj/dfLinSi (Ax) (no source held here)

- Data object Logical/Simulation/Motion/gkLinSobj/gkLinSa (Apt) (no source held here)

- Data object Logical/Simulation/Motion/gkLinSobj/gkLinSi (Ax) (no source held here)

- Data object Logical/Simulation/Motion/fwRotSobj/fwRotSa (Apt) (no source held here)

- Data object Logical/Simulation/Motion/fwRotSobj/fwRotSi (Ax) (no source held here)

- Data object Logical/Simulation/Motion/mdRotSobj/mdRotSa (Apt) (no source held here)

- Data object Logical/Simulation/Motion/mdRotSobj/mdRotSi (Ax) (no source held here)

- Data object Logical/Simulation/Motion/fwLinSobj/fwLinSa (Apt) (no source held here)

- Data object Logical/Simulation/Motion/fwLinSobj/fwLinSi (Ax) (no source held here)

- Data object Logical/Simulation/Motion/mdLinSobj/mdLinSa (Apt) (no source held here)

- Data object Logical/Simulation/Motion/mdLinSobj/mdLinSi (Ax) (no source held here)

### Program Logical/Simulation/Technology/simulation (ANSIC) - Roman Parák program for simulation.

#### simulation.c - Init, cyclic, exit code
```c
/*********************************************************************************************
* B&R Automation - Perfection in Automation (https://www.br-automation.com)
    ******************************************************************************************
    * Program 	    : Master's Thesis - Soccer Table (Simulation)
    * Author  	    : Roman Parak
    * Created 	    : date ...
	* University    : Brno University of Technology(BUT)
	* Faculty       : Faculty of Mechanical Engineering(FME)
	* Study Program : Applied Computer Science and Control
	* Institute     : Institute of Automation and Computer Science
**********************************************************************************************
* Implementation OF PROGRAM simulation(Simulation/Technology/simulation/Program/simulation.c)
**********************************************************************************************/

/*************************** LIBRARIES *********************************/
#include <bur/plc.h>
#include <bur/plctypes.h>
#include <astime.h>
#include <math.h>

#include "rp_funcx1.h"
#include "Structures/simulation_str.h"
#include "Functions/sim_mapp.h"

#ifdef _DEFAULT_INCLUDES
	#include <AsDefault.h>
#endif

/*************************** DEFINITIONS *******************************/
#define EACH_FORMATION 1;

/************************ LOCAL VARIABLES ******************************/

// struct - rp_funcx1
_LOCAL struct forecast_direction f_d;
_LOCAL struct calculation_posDummies c_ppd;
_LOCAL struct calculation_crossingBall c_cb[2];
_LOCAL struct calculation_displacementOfAxes c_doa;
_LOCAL struct start_rotaryAxis start_rotaryAxis_0;
_LOCAL struct control_temperature c_temp;
_LOCAL struct axes_control axes_control_0[4];
_LOCAL struct ball_shooting ball_s;
_LOCAL struct check_attack_mode check_attack_mode_0;
_LOCAL struct start_virtualAxis s_virtualA;
// struct - MpAlarmX
_LOCAL MpAlarmXListUIConnectType AlarmListUI_ConnectType;
_LOCAL MpAlarmXHistoryUIConnectType AlarmHistoryUI_ConnectType;
// udint
_LOCAL UDINT alarm_device_address, specific_directionOfBall;
// usint
_LOCAL USINT max_numberOfFormation;
_LOCAL USINT i_axisNum;
_LOCAL USINT i_bs;
_LOCAL USINT i_ppd, i_ccd, i_ccdCPU, i_ccdHUM, i_cdoa1, i_cdoa2, i_cdoa3;
_LOCAL USINT c_dp;
_LOCAL USINT i_def, i_dp1, i_dp2;
_LOCAL USINT c_bState;
// bool
_LOCAL BOOL ESTOP,error_s,reset_safetyESTOP;
_LOCAL BOOL start_game;
// real
_LOCAL REAL x_posOfCPU[4];
_LOCAL REAL x_posOfHUM[4];
// OUPTUT from the SENSOR & CAMERA
_LOCAL REAL ball1[2], ball2[2], time_B2B;
_LOCAL REAL optical_sensor[4];
_LOCAL REAL reflex_sensor[4];
// state machine
_LOCAL soccer_table_ENUM SOCCER_TABLE_STEP;
_LOCAL soccer_table_ENUM BEFORE_STATE;

/**********************************************************************************************************/
/********************************************** INIT PROGRAM **********************************************/
/**********************************************************************************************************/
void _INIT ProgramInit(void)
{
    /*********************************** declaration variables **********************************/
    // generally
    max_numberOfFormation = 4;
    // axis type -> MAPP
    // linear
	gLinkAxes_linear[0] = gk_mappAxisLS;
    gLinkAxes_linear[1] = df_mappAxisLS;
    gLinkAxes_linear[2] = md_mappAxisLS;
    gLinkAxes_linear[3] = fw_mappAxisLS;
    // rotary
    gLinkAxes_rotary[0] = gk_mappAxisRS;
    gLinkAxes_rotary[1] = df_mappAxisRS;
    gLinkAxes_rotary[2] = md_mappAxisRS;
    gLinkAxes_rotary[3] = fw_mappAxisRS;

    /************************************ control of AlarmX ************************************/
    // adjustment device name
    alarm_device_address = (UDINT) strcpy(mp_alarmX.deviceName_no1_exp,"EXPORT_HISTORY");
    // MpAlarmX Core
    mp_alarmX.mp_core.MpLink         = &gAlarmXCoreS;
    mp_alarmX.mp_core.Enable         = 1;
    // MpAlarmX ListUI
    mp_alarmX.mp_listUI.MpLink       = &gAlarmXCoreS;
    mp_alarmX.mp_listUI.Enable       = 1;
    mp_alarmX.mp_listUI.UIConnect    = &AlarmListUI_ConnectType;
    // MpAlarmX History
    mp_alarmX.mp_history.MpLink      = &gAlarmXHistoryS;
    mp_alarmX.mp_history.Enable      = 1;
    mp_alarmX.mp_history.DeviceName  = &mp_alarmX.deviceName_no1_exp;
    // MpAlarmX HistoryUI
    mp_alarmX.mp_historyUI.MpLink    = &gAlarmXHistoryS;
    mp_alarmX.mp_historyUI.Enable    = 1;
    mp_alarmX.mp_historyUI.UIConnect = &AlarmHistoryUI_ConnectType;

    /************************************* control of axes **************************************/
    for(i_axisNum = 0; i_axisNum <= max_numberOfFormation - 1; i_axisNum++){
        // initialization ACOPOS variables through function(get_axisParam), that returns two variables type of UDINT
        // into the structure -> axesAcopos(have two parameters : linear, rotary)
        axis_acopos = get_axisParam(i_axisNum);
        // linear -> LinMot
        // linear axis basic
        mp_Axis.mp_axisLinear[i_axisNum].Enable     = 1;
        mp_Axis.mp_axisLinear[i_axisNum].MpLink     = &gLinkAxes_linear[i_axisNum];
        mp_Axis.mp_axisLinear[i_axisNum].Parameters = &mp_Axis.param_axisLinear[i_axisNum];
        mp_Axis.mp_axisLinear[i_axisNum].Axis       = axis_acopos.linear;
        // linear cyclic set
        mp_Axis.mp_cyclicSetLinear[i_axisNum].Enable     = 1;
        mp_Axis.mp_cyclicSetLinear[i_axisNum].MpLink     = &gLinkAxes_linear[i_axisNum];
        mp_Axis.mp_cyclicSetLinear[i_axisNum].Parameters = &mp_Axis.param_cyclicSetLinear[i_axisNum];
		// adjustment max velocity
		mp_Axis.param_cyclicSetLinear[i_axisNum].PositionModeMaxVelocity = 30000;
		// config
		mp_Axis.mp_configAxisLinear[i_axisNum].Enable 		 = 1;
		mp_Axis.mp_configAxisLinear[i_axisNum].MpLink 		 = &gLinkAxes_linear[i_axisNum];
		mp_Axis.mp_configAxisLinear[i_axisNum].Configuration = &mp_Axis.param_configAxisLinear[i_axisNum];
        // rotary -> EnDat
        // rotary axis basic
        mp_Axis.mp_axisRotary[i_axisNum].Enable     = 1;
        mp_Axis.mp_axisRotary[i_axisNum].MpLink     = &gLinkAxes_rotary[i_axisNum];
        mp_Axis.mp_axisRotary[i_axisNum].Parameters = &mp_Axis.param_axisRotary[i_axisNum];
        mp_Axis.mp_axisRotary[i_axisNum].Axis       = axis_acopos.rotary;
        // rotary cyclic set
        mp_Axis.mp_cyclicSetRotary[i_axisNum].Enable     = 1;
        mp_Axis.mp_cyclicSetRotary[i_axisNum].MpLink     = &gLinkAxes_rotary[i_axisNum];
        mp_Axis.mp_cyclicSetRotary[i_axisNum].Parameters = &mp_Axis.param_cyclicSetRotary[i_axisNum];
		// adjustment max velocity
		mp_Axis.param_cyclicSetRotary[i_axisNum].PositionModeMaxVelocity = 85000;
		// config
		mp_Axis.mp_configAxisRotary[i_axisNum].Enable 		 = 1;
		mp_Axis.mp_configAxisRotary[i_axisNum].MpLink 		 = &gLinkAxes_rotary[i_axisNum];
		mp_Axis.mp_configAxisRotary[i_axisNum].Configuration = &mp_Axis.param_configAxisRotary[i_axisNum];
		// temperature - linear
		mp_Axis.param_axisLinear[i_axisNum].CyclicRead.MotorTempMode = mpAXIS_READ_POLLING_5s;
		// temperature - rotary
		mp_Axis.param_axisRotary[i_axisNum].CyclicRead.MotorTempMode = mpAXIS_READ_POLLING_5s;
    }
    // initialization switch
    SOCCER_TABLE_STEP = RST_EMPTY;
    // initialization x axes for CPU
    x_posOfCPU[0] = 800;
    x_posOfCPU[1] = 2300;
    x_posOfCPU[2] = 5300;
    x_posOfCPU[3] = 8300;
    // initialization x axes for HUMAN
    x_posOfHUM[0] = 3800;
    x_posOfHUM[1] = 6800;
    x_posOfHUM[2] = 9800;
    x_posOfHUM[3] = 11300;
    // OUPTUT from the SENSOR & CAMERA
    // CAMERA
    ball1[0] = 0;
    ball1[1] = 0;
    ball2[0] = 0;
    ball2[1] = 0;
    time_B2B = 0;
    // SENSOR
    optical_sensor[0] = 0;
    optical_sensor[1] = 0;
    optical_sensor[2] = 0;
    optical_sensor[3] = 0;

    reflex_sensor[0] = 1;
    reflex_sensor[1] = 1;
    reflex_sensor[2] = 1;
    reflex_sensor[3] = 1;
	// init safety
	ESTOP = 1;
	// axes control
	// FB for linear and fotary axes -> Control
	axes_control_0[0].Enable			 = 1;
	axes_control_0[0].linear_axis_cyclic = &mp_Axis.mp_cyclicSetLinear[0];
	axes_control_0[0].linear_axis_param  = &mp_Axis.param_cyclicSetLinear[0];
	axes_control_0[0].rotary_axis_cyclic = &mp_Axis.mp_cyclicSetRotary[0];
	axes_control_0[0].rotary_axis_param  = &mp_Axis.param_cyclicSetRotary[0];

	s_virtualA.Enable 	  = 1;
	s_virtualA.axis_name  = &mp_Axis.mp_axisLinear[0];
	s_virtualA.axis_param = &mp_Axis.param_axisLinear[0];
}// end _INIT

/**********************************************************************************************************/
/********************************************** MAIN PROGRAM **********************************************/
/**********************************************************************************************************/
void _CYCLIC ProgramCyclic(void)
{
    switch(SOCCER_TABLE_STEP){
		case RST_EMPTY:
			{

			}
			break;
		case RST_INITIALIZATION_1:
			{
				// home virtual linear axis
				s_virtualA.start_btn = 1;
				start_virtualAxis(&s_virtualA);

				if(s_virtualA.succesfully == 1 && (mp_Axis.mp_axisLinear[0].PowerOn == 1 && mp_Axis.mp_axisLinear[0].IsHomed == 1)){
					SOCCER_TABLE_STEP = RST_INITIALIZATION_2;
				}
			}
			break;
		case RST_INITIALIZATION_2:
			{

			}
			break;
		case RST_INITIALIZATION_3:
			{

			}
			break;
		case RST_INITIALIZATION_4:
			{
				check_attack_mode_0.ball1_x = ball1[0];
				check_attack_mode_0.ball1_y = ball1[1];
				check_attack_mode_0.ball2_x = ball2[0];
				check_attack_mode_0.ball2_y = ball2[1];

				check_attack_mode_0.act_displacement_cpu[2] = 112;
				check_attack_mode_0.angle_ofRotation[2]     = -250;
				// call function
				check_attack_mode(&check_attack_mode_0);
			}
			break;
        case RST_CALCULATION_DEFENSE:
            {
                // calculation forecast direction
                f_d.ball1_x = ball1[0];
                f_d.ball1_y = ball1[1];
                f_d.ball2_x = ball2[0];
                f_d.ball2_y = ball2[1];
                forecast_direction(&f_d);
                // calculation pos dummies opponent
				// maximum displacement of individual axes
				c_ppd.max_disp[0] = 1000;
				c_ppd.max_disp[0] = 1850;
				c_ppd.max_disp[0] = 650;
				c_ppd.max_disp[0] = 955;
				// minimum displacement of individual axes
				c_ppd.min_disp[0] = -1000;
				c_ppd.min_disp[0] = -1850;
				c_ppd.min_disp[0] = -650;
				c_ppd.min_disp[0] = -955;
                for(i_ppd = 0; i_ppd < (int)(sizeof(optical_sensor)/sizeof(optical_sensor[0])); i_ppd++){
                    c_ppd.displacement[i_ppd] = optical_sensor[i_ppd];
                }

                calculation_posDummies(&c_ppd);
                // calculation crossing ball
                for(i_ccd = 0; i_ccd < (int)(sizeof(ball1)/sizeof(ball1[0])); i_ccd++){
                    c_cb[i_ccd].ball1_x = ball1[0];
                    c_cb[i_ccd].ball1_y = ball1[1];
                    c_cb[i_ccd].ball2_x = ball2[0];
                    c_cb[i_ccd].ball2_y = ball2[1];
                    c_cb[i_ccd].first_reflection_x  = f_d.first_reflectionX;
                    c_cb[i_ccd].first_reflection_y  = f_d.first_reflectionY;
                    c_cb[i_ccd].second_reflection_x = f_d.second_reflectionX;
                    c_cb[i_ccd].second_reflection_y = f_d.second_reflectionY;
                    c_cb[i_ccd].tilted   = f_d.tilted;
                    c_cb[i_ccd].time_B2B = time_B2B;

                    if(i_ccd == 0){
                        for(i_ccdCPU = 0; i_ccdCPU < (int)(sizeof(x_posOfCPU)/sizeof(x_posOfCPU[0])); i_ccdCPU++){
                            c_cb[i_ccd].x_positions[i_ccdCPU] = x_posOfCPU[i_ccdCPU];
                        }
                    }else if(i_ccd == 1){
                        for(i_ccdHUM = 0; i_ccdHUM < (int)(sizeof(x_posOfHUM)/sizeof(x_posOfHUM[0])); i_ccdHUM++){
                            c_cb[i_ccd].x_positions[i_ccdHUM] = x_posOfHUM[i_ccdHUM];
                        }
                    }
                    calculation_crossingBall(&c_cb[i_ccd]);
                }
                // calculation displacement
                c_doa.tilted             = f_d.tilted;
                specific_directionOfBall = (UDINT) strcpy(c_doa.specific_direction,f_d.specific_direction);
                for(i_cdoa1 = 0; i_cdoa1 < (int)(sizeof(c_cb[1].count_axesIntersection)/sizeof(c_cb[1].count_axesIntersection[0])); i_cdoa1++){
                    c_doa.count_axesIntersectionHUM[i_cdoa1] = c_cb[1].count_axesIntersection[i_cdoa1];
                }
                for(i_cdoa2 = 0; i_cdoa2 < (int)(sizeof(c_cb[0].act_posOfAxesY)/sizeof(c_cb[0].act_posOfAxesY[0])); i_cdoa2++){
                    c_doa.act_posOfAxesCPU_Y[i_cdoa2]    = c_cb[0].act_posOfAxesY[i_cdoa2];
                    c_doa.time_axisIntersection[i_cdoa2] = c_cb[0].time_axisIntersection[i_cdoa2];
                    c_doa.act_displacementCPU[i_cdoa2]   = 0; // actual displacement
                    c_doa.reversed_HUM[i_cdoa2]          = reflex_sensor[i_cdoa2];
                }
                c_doa.act_posOfAxesHUM_Y[0] = c_cb[1].act_posOfAxesY[3];
                c_doa.act_posOfAxesHUM_Y[1] = c_cb[1].act_posOfAxesY[2];
                c_doa.act_posOfAxesHUM_Y[2] = c_cb[1].act_posOfAxesY[1];
                c_doa.act_posOfAxesHUM_Y[3] = c_cb[1].act_posOfAxesY[0];
                for(i_cdoa3 = 0; i_cdoa3 < (int)(sizeof(c_ppd.actual_positionsOfDummies)/sizeof(c_ppd.actual_positionsOfDummies[0])); i_cdoa3++){
                    c_doa.act_posOfDummiesH[i_cdoa3] = c_ppd.actual_positionsOfDummies[i_cdoa3];
                }
                c_doa.x_posOfBall[0] = ball1[0];
                c_doa.x_posOfBall[1] = ball2[0];
                calculation_displacementOfAxes(&c_doa);

				for(i_def = 0; i_def <= max_numberOfFormation - 1; i_def++){
					if(!isnan(c_doa.velocity[i_def])){
						axes_control_0[i_def].linear_param.acceleration = c_doa.acceleration[i_def];
						axes_control_0[i_def].linear_param.deceleration = c_doa.deceleration[i_def];
						axes_control_0[i_def].linear_param.velocity     = c_doa.velocity[i_def];
						axes_control_0[i_def].linear_param.displacement = c_doa.displacement[i_def];
					}
				}

				/*
				if(ESTOP == 0){
					SOCCER_TABLE_STEP = RST_SAFETY;
				}else{
					c_dp = 0;

					if(c_dp == 0){
						SOCCER_TABLE_STEP = RST_MOVE_INTO_DEFENSE_POS1;
					}
				}
				*/
            }
            break;
		case RST_MOVE_INTO_DEFENSE_POS1:
			{
				for(i_dp1 = 0; i_dp1 <= max_numberOfFormation - 1; i_dp1++){
					axes_control_0[i_dp1].start_move = 1;
				}

				if(ESTOP == 0){
					SOCCER_TABLE_STEP = RST_SAFETY;
				}else{
					SOCCER_TABLE_STEP = RST_MOVE_INTO_DEFENSE_POS2;
				}
			}
			break;
		case RST_MOVE_INTO_DEFENSE_POS2:
			{
				for(i_dp2 = 0; i_dp2 <= max_numberOfFormation - 1; i_dp2++){
					if(axes_control_0[i_dp2].successfully == 1){
						axes_control_0[i_dp2].start_move = 0;
						c_dp++;
					}
				}

				if(ESTOP == 0){
					SOCCER_TABLE_STEP = RST_SAFETY;
				}else{
					if(c_dp == max_numberOfFormation){
						SOCCER_TABLE_STEP = RST_INITIALIZATION_4;
					}
				}
			}
		case RST_SAFETY:
			{
			}
			break;
		case RST_AFTER_SAFETY:
			{

			}
			break;
    }// end switch

    /************************** call function & function blocks **************************/
    // AlarmX
    MpAlarmXCore(&mp_alarmX.mp_core);
    MpAlarmXListUI(&mp_alarmX.mp_listUI);
    MpAlarmXHistory(&mp_alarmX.mp_history);
    MpAlarmXHistoryUI(&mp_alarmX.mp_historyUI);
    // Active AxisBasic & AxisCyclicSet -> through the individual functions
    start_axesBasic(max_numberOfFormation,&mp_Axis.mp_axisLinear,&mp_Axis.mp_axisRotary);
    start_axesCyclic(max_numberOfFormation,&mp_Axis.mp_cyclicSetLinear,&mp_Axis.mp_cyclicSetRotary);

	// control temperature
	//control_temperature(&c_temp);
	if(SOCCER_TABLE_STEP >= 3){
		axes_control(&axes_control_0[0]);
	}

}// end _CYCLIC
```

#### simulation_str.h
```c
/*********************************************************************************************
* B&R Automation - Perfection in Automation (https://www.br-automation.com)
    ******************************************************************************************
    * Program 	    : Master's Thesis - Soccer Table (Simulation)
    * Author  	    : Roman Parak
    * Created 	    : date ...
	* University    : Brno University of Technology(BUT)
	* Faculty       : Faculty of Mechanical Engineering(FME)
	* Study Program : Applied Computer Science and Control
	* Institute     : Institute of Automation and Computer Science
**********************************************************************************************
* Implementation OF PROGRAM simulation(Simulation/Technology/simulation/Structures/simulation_str.h)
**********************************************************************************************/

/*************************** LIBRARIES *********************************/
#include <bur/plc.h>
#include <bur/plctypes.h>
#include <AsString.h>
#include <AsWStr.h>

#ifdef _DEFAULT_INCLUDES
    #include <AsDefault.h>
#endif

/**********************************************************************************************************/
/************************************** STRUCTURE TYPE ****************************************************/
/**********************************************************************************************************/

/***************************************** sim_mapp.h *****************************************************/
/***************************** ALARM ***********************************/
typedef struct mappAlarmX_STR{
    // list
    struct MpAlarmXCore   mp_core;
    struct MpAlarmXListUI mp_listUI;
    // history
    struct    MpAlarmXHistory mp_history;
    struct    MpAlarmXHistoryUI mp_historyUI;
    plcstring deviceName_no1_exp[21];
} mappAlarmX_STR;

/***************************** AXIS ************************************/
typedef struct mappAxisBasic_STR{
	// === Linear Axes === //
	// axis basic
	struct MpAxisBasic        mp_axisLinear[4];
	struct MpAxisBasicParType param_axisLinear[4];
	// cyclic set
	struct MpAxisCyclicSet        mp_cyclicSetLinear[4];
	struct MpAxisCyclicSetParType param_cyclicSetLinear[4];
	// config
	struct MpAxisBasicConfig mp_configAxisLinear[4];
	struct MpAxisBasicConfigType param_configAxisLinear[4];
	// === Rotary Axes === //
	// axis basic
	struct MpAxisBasic        mp_axisRotary[4];
	struct MpAxisBasicParType param_axisRotary[4];
	// cyclic set
	struct MpAxisCyclicSet        mp_cyclicSetRotary[4];
	struct MpAxisCyclicSetParType param_cyclicSetRotary[4];
	// config
	struct MpAxisBasicConfig mp_configAxisRotary[4];
	struct MpAxisBasicConfigType param_configAxisRotary[4];
} mappAxisBasic_STR;

/***************************** GET AXIS PARAM. ************************************/
typedef struct axesAcopos{
    UDINT linear;
    UDINT rotary;
}axesAcopos;

/*********************************** sim_forecast_direction.h *********************************************/
/***************************** FORECAST DIR.. ************************************/
typedef struct forecastDirection{
	BOOL direction;
	INT first_reflectX;
	INT first_reflectY;
	INT second_reflectX;
	INT second_reflectY;
	plcstring specific_direction[30];
}forecastDirection;
/***************************** CALC. DIR. OF TILT **********************************/
typedef struct tiltDirection{
	INT first_reflectX;
	INT first_reflectY;
	INT state_ofDirection;
    plcstring specific_direction[10];
}tiltDirection;
/***************************** CALC. NEXT DIR. *************************************/
typedef struct nextDirection{
	INT second_reflectX;
	INT second_reflectY;
}nextDirection;

/**********************************************************************************************************/
/**************************************** GLOBAL VARIABLES ************************************************/
/**********************************************************************************************************/

/***************************************** sim_mapp.h *****************************************************/
// my structures
_GLOBAL mappAlarmX_STR mp_alarmX;
_GLOBAL mappAxisBasic_STR mp_Axis;
_GLOBAL axesAcopos axis_acopos;

// axis type -> ACOPOS
// goalkeeper
_GLOBAL ACP10AXIS_typ gkLinS;
_GLOBAL ACP10AXIS_typ gkRotS;
// defender
_GLOBAL ACP10AXIS_typ dfLinS;
_GLOBAL ACP10AXIS_typ dfRotS;
// midfielder
_GLOBAL ACP10AXIS_typ mdLinS;
_GLOBAL ACP10AXIS_typ mdRotS;
// forward
_GLOBAL ACP10AXIS_typ fwLinS;
_GLOBAL ACP10AXIS_typ fwRotS;
// axis type -> MAPP
_GLOBAL struct MpComIdentType gLinkAxes_rotary[4];
_GLOBAL struct MpComIdentType gLinkAxes_linear[4];

/**********************************************************************************************************/
/************************************** FUNCTIONS & FUNCTIONS BLOCKS **************************************/
/**********************************************************************************************************/
void start_axesBasic(USINT num_ofAxes,struct MpAxisBasic* axis_linear,struct MpAxisBasic* axis_rotary);
void start_axesCyclic(USINT num_ofAxes,struct MpAxisCyclicSet* cyclic_linear,struct MpAxisCyclicSet* cyclic_rotary);
struct axesAcopos get_axisParam(int idx_ofIteration);
```

#### sim_mapp.h
```c
/*********************************************************************************************
* B&R Automation - Perfection in Automation (https://www.br-automation.com)
    ******************************************************************************************
    * Program 	    : Master's Thesis - Soccer Table (Simulation)
    * Author  	    : Roman Parak
    * Created 	    : date ...
	* University    : Brno University of Technology(BUT)
	* Faculty       : Faculty of Mechanical Engineering(FME)
	* Study Program : Applied Computer Science and Control
	* Institute     : Institute of Automation and Computer Science
**********************************************************************************************
* Implementation OF PROGRAM simulation(Simulation/Technology/simulation/Functions/sim_mapp.h)
**********************************************************************************************/

/*************************** LIBRARIES *********************************/
#include <bur/plc.h>
#include <bur/plctypes.h>
#include <AsString.h>
#include <AsWStr.h>

#ifdef _DEFAULT_INCLUDES
    #include <AsDefault.h>
#endif

/**********************************************************************************************************/
/************************************** FUNCTIONS & FUNCTIONS BLOCKS **************************************/
/**********************************************************************************************************/
void start_axesBasic(USINT num_ofAxes,struct MpAxisBasic* axis_linear,struct MpAxisBasic* axis_rotary){
    int i;
    // Axis Basic
    // function to start the individual axes
    // the cycle is carried out through number of axes
    for(i = 0; i <= num_ofAxes - 1; i++){
        // mapp axis basic
        MpAxisBasic(&axis_linear[i]);
        MpAxisBasic(&axis_rotary[i]);
    }
}

void start_axesCyclic(USINT num_ofAxes,struct MpAxisCyclicSet* cyclic_linear,struct MpAxisCyclicSet* cyclic_rotary){
    int i;
    // Axis Cyclic Set
    // function to start the individual axes
    // the cycle is carried out through number of axes
    for(i = 0; i <= num_ofAxes - 1; i++){
        // mapp axis cyclic set
        MpAxisCyclicSet(&cyclic_linear[i]);
        MpAxisCyclicSet(&cyclic_rotary[i]);
    }
}

struct axesAcopos get_axisParam(int idx_ofIteration){
    // input into the function is number of iteration(in the init part)
    // create auxiliary structures and enumeration type(for state machine)
    struct axesAcopos a;
    typedef enum {aNUM1 = 0, aNUM2, aNUM3, aNUM4}wState_ofAxes;
    wState_ofAxes new_idx; // initialize state machine
    new_idx = idx_ofIteration;
    // gradually into the state machine loading indexes from initialization part
    // each state of machine has initialization both engines linear and rotary, on its own axis
    // output of this function is structure, that has two parameters(linear,rotary axis)
    switch(new_idx){
        case aNUM1:
            // goalkeeper
            a.linear = &gkLinearA;
            a.rotary = &gkRotaryA;
            return a;
            break;
        case aNUM2:
            // defender
            a.linear = &dfLinearB;
            a.rotary = &dfRotaryB;
            return a;
            break;
        case aNUM3:
            // midfielder
            a.linear = &mdLinearC;
            a.rotary = &mdRotaryC;
            return a;
            break;
        case aNUM4:
            // forward
            a.linear = &fwLinearD;
            a.rotary = &fwRotaryD;
            break;
    }
}
```

### Program Logical/Simulation/Technology/sim_cam_sens_sd_s (ANSIC) - Lubo,Radek program for simulation.

#### main_sim.c - Init, cyclic, exit code
```c
/*********************************************************************************************
* B&R Automation - Perfection in Automation (https://www.br-automation.com)
    ******************************************************************************************
    * Program 	    : Bachelor's Thesis
    * Author  	    : Lubo Bubco, Radek Otradovský
    * Created 	    : date ...
	* University    : Brno University of Technology(BUT)
	* Faculty       : Faculty of Mechanical Engineering(FME), Faculty of Electrical Engineering and Communication(FEEC)
**********************************************************************************************
* Implementation OF PROGRAM sim_cam_sens_sd_s(Simulation/Technology/sim_cam_sens_sd_s/main_sim.c)
**********************************************************************************************/

#include <bur/plctypes.h>
#include <string.h>
#include <math.h>
#include "rp_funcx1.h"

#ifdef _DEFAULT_INCLUDES
	#include <AsDefault.h>
#endif

_LOCAL struct measurement_ofScore measurement_ofScore_0;

void _INIT ProgramInit(void)
{

}

void _CYCLIC ProgramCyclic(void)
{
    measurement_ofScore(&measurement_ofScore_0);
}
```

### Program Logical/Real_Game/Technology/table_football (ANSIC) - Roman Parák program for real game.

#### mapp.h
```c
/*********************************************************************************************
* B&R Automation - Perfection in Automation (https://www.br-automation.com)
    ******************************************************************************************
    * Program 	    : Master's Thesis - Soccer Table (Table Football - real game)
    * Author  	    : Roman Parak
    * Created 	    : date ...
	* University    : Brno University of Technology(BUT)
	* Faculty       : Faculty of Mechanical Engineering(FME)
	* Study Program : Applied Computer Science and Control
	* Institute     : Institute of Automation and Computer Science
**********************************************************************************************
* Implementation OF PROGRAM table_football(Real_Game/Technolog/table_football/Functions/mapp.h)
**********************************************************************************************/

/*************************** LIBRARIES *********************************/
#include <bur/plc.h>
#include <bur/plctypes.h>
#include <AsString.h>
#include <standard.h>
#include <AsWStr.h>
#include <stdio.h>
#include <math.h>

#ifdef _DEFAULT_INCLUDES
    #include <AsDefault.h>
#endif

/**********************************************************************************************************/
/************************************** FUNCTIONS & FUNCTIONS BLOCKS **************************************/
/**********************************************************************************************************/
void start_axesBasic(USINT num_ofAxes,struct MpAxisBasic* axis_linear,struct MpAxisBasic* axis_rotary){
    int i;
    // Axis Basic
    // function to start the individual axes
    // the cycle is carried out through number of axes
    for(i = 0; i <= num_ofAxes - 1; i++){
        // mapp axis basic
        MpAxisBasic(&axis_linear[i]);
        MpAxisBasic(&axis_rotary[i]);
    }
}

void start_axesCyclic(USINT num_ofAxes,struct MpAxisCyclicSet* cyclic_linear,struct MpAxisCyclicSet* cyclic_rotary){
    int i;
    // Axis Cyclic Set
    // function to start the individual axes
    // the cycle is carried out through number of axes
    for(i = 0; i <= num_ofAxes - 1; i++){
        // mapp axis cyclic set
        MpAxisCyclicSet(&cyclic_linear[i]);
        MpAxisCyclicSet(&cyclic_rotary[i]);
    }
}

struct axesAcopos get_axisParam(int idx_ofIteration){
    // input into the function is number of iteration(in the init part)
    // create auxiliary structures and enumeration type(for state machine)
    struct axesAcopos a;
    typedef enum {aNUM1 = 0, aNUM2, aNUM3, aNUM4}wState_ofAxes;
    wState_ofAxes new_idx; // initialize state machine
    new_idx = idx_ofIteration;
    // gradually into the state machine loading indexes from initialization part
    // and this run the function blocks
    // each state of machine has initialization both engines linear and rotary, on its own axis
    // output of this function is structure, that has two parameters(linear,rotary axis)
    switch(new_idx){
        case aNUM1:
            // goalkeeper
            a.linear = &linGK;
            a.rotary = &rotGK;
            return a;
            break;
        case aNUM2:
            // defender
            a.linear = &linDF;
            a.rotary = &rotDF;
            return a;
            break;
        case aNUM3:
            // midfielder
            a.linear = &linearMD;
            a.rotary = &rotaryMD;
            return a;
            break;
        case aNUM4:
            // forward
            a.linear = &linearFW;
            a.rotary = &rotaryFW;
			return a;
            break;
    }
}

void start_cs(USINT num_ofAxes,struct MpAxisCyclicSet* cyclic_linear,struct MpAxisCyclicSet* cyclic_rotary){

	switch(num_ofAxes){
		case 1:
			{
				cyclic_linear[0].CyclicPosition = 1;
				cyclic_rotary[0].CyclicPosition = 1;
			}
			break;
		case 2:
			{
				cyclic_linear[0].CyclicPosition = 1;
				cyclic_linear[1].CyclicPosition = 1;
				cyclic_rotary[0].CyclicPosition = 1;
				cyclic_rotary[1].CyclicPosition = 1;

			}
			break;
		case 3:
			{
				cyclic_linear[0].CyclicPosition = 1;
				cyclic_linear[1].CyclicPosition = 1;
				cyclic_linear[2].CyclicPosition = 1;
				cyclic_rotary[0].CyclicPosition = 1;
				cyclic_rotary[1].CyclicPosition = 1;
				cyclic_rotary[2].CyclicPosition = 1;
			}
			break;
		case 4:
			{
				cyclic_linear[0].CyclicPosition = 1;
				cyclic_linear[1].CyclicPosition = 1;
				cyclic_linear[2].CyclicPosition = 1;
				cyclic_linear[3].CyclicPosition = 1;
				cyclic_rotary[0].CyclicPosition = 1;
				cyclic_rotary[1].CyclicPosition = 1;
				cyclic_rotary[2].CyclicPosition = 1;
				cyclic_rotary[3].CyclicPosition = 1;
			}
			break;
	}// end switch

}
```

#### Program Logical/Real_Game/Technology/table_football/Program
